# EPICS autosave request: iocBoot/iocxxx/vxWorks/pf4common.req
$(P)$(H)E:local
$(P)$(H)useMono
$(P)$(H)filterAl.EGU
$(P)$(H)filterTi.EGU
$(P)$(H)filterGlass.EGU
